Staubli VAL3: sampleGripping.pgx

program sampleGripping(bool gripSample (dimensions=1), string command (dimensions=1), num sio_ID (dimensions=1))
  local jointRx pickingPosJoint
  local pointRx pickingPosPoint
  local string reply
begin
  //**************************************************
  // Method to take or place sample at the magazine or at the spinner.
  // The former is determined by the gripSample argument. The latter
  // is determined from the position (herej()) of the arm when this
  // method is called.
  //**************************************************

  // For picking samples (we end with sample in the gripper), we must have an open
  // gripper to start with
  if (gripSample==true) and (switchGripper==true)
    switchGripper=false
  else
  endIf

  // The current pick position is either the currentSamPosJ or spinnerPosition
  // We don't know which and to make this flexible we set for the scope of this method
  pickingPosJoint=herej()
  pickingPosPoint=jointToPoint(flange,world,pickingPosJoint)
  // Move in to the sample
  movel(appro(pickingPosPoint,{0,0,80,0,0,0}),flange,mNomSpeed)
  waitEndMove()

  // Grab the sample and move out
  switchGripper=gripSample
  movel(appro(pickingPosPoint,{0,0,0,0,0,0}),flange,mNomSpeed)
  waitEndMove()

  reply=command+":done"
  taskCreate "sendStatus",10,sendStatus(reply,sio_ID)
  taskKill("sampleGripping")

end
